{attribute 'qualified_only'}
VAR_GLOBAL
	stComponents			: ST_Components;
	stComponentsView		: ST_Components_HMI_View;
	stComponentsCmd			: ST_Components_HMI_Command;
	stControl				: ST_ControlElements;
	stGroup					: ST_GroupElements;
	stTop					: ST_TopElements;
END_VAR

(* stored: Version 1.1.0.1
   GVL GVL_Elements: Id {4de1326c-c6ad-0262-2ca0-1f3e691aed53} *)
